// TIA Portal project "Donanım_Kesmesi_Uygulaması_V1" (V16)
// Vorlageprojekt für das Buch mit Zielsystem S7-1200

(* hardware
DEVICE "S7-1200-Station_1"  S7-1200 Station
   slot 0: "Baugruppenträger_0"  Rack  V1.0
   slot 1: "PLC_1"  CPU 1214C DC/DC/DC  6ES7 214-1AG40-0XB0  V4.4
   slot 2: "DQ 16x24VDC_1"  SM 1222 DQ16 x 24VDC  6ES7 222-1BH32-0XB0  V2.0
   slot 3: "AQ 2x14BIT_1"  SM 1232 AQ2  6ES7 232-4HB32-0XB0  V2.1
*)

// ===== PLC "PLC_1"  CPU 1214C DC/DC/DC =====

VAR_GLOBAL   // PLC tag table "Standard-Variablentabelle"
   "Sistem_Start_Mem." AT %M10.0 : Bool;
   "Kenar_Darbesi_1" AT %M20.0 : Bool;
   "Kenar_Darbesi_2" AT %M20.1 : Bool;
   "Kenar_Darbesi_3" AT %M20.2 : Bool;
   "Ürün_Sayısı" AT %MW30 : Int;
END_VAR

VAR_GLOBAL   // PLC tag table "Inputs"
   "Start_But" AT %I0.0 : Bool;
   "Stop_But" AT %I0.1 : Bool;
   "Acil_Stop_But" AT %I0.2 : Bool;
   "Sensör_!" AT %I0.3 : Bool;
   "Sensör_2" AT %I0.4 : Bool;
   "Sensör_3" AT %I0.5 : Bool;
END_VAR

VAR_GLOBAL   // PLC tag table "Outputs"
   "Durdurma_Kanalı" AT %Q0.0 : Bool;
   "Sayıcı_Ekranı" AT %QW30 : Int;
   "Konveyör_1" AT %QW32 : Int;
   "Konveyör_2" AT %QW34 : Int;
END_VAR

// folder: System blocks/Program resources

DATA_BLOCK "Tımer_1"   // DB1
{ S7_Optimized_Access := 'TRUE' }
AUTHOR : Simatic
FAMILY : IEC
NAME : IEC_TMR
VERSION : 1.0
// stored: InstanceOfName IEC_TIMER
"IEC_TIMER"
BEGIN
END_DATA_BLOCK

// folder: (top level)

FUNCTION "MHJ-PLC-Lab-Function-S71200" : Void   // FC9000, SCL
{ S7_Optimized_Access := 'TRUE' }
VERSION : 0.1
   VAR_TEMP
      rdTimeReturn : Int;
      outputTime : DTL;
      SyncVal : Byte;
      forVal : Int;
      forVal_2 : Int;
      Value : Byte;
   END_VAR
   VAR CONSTANT
      CompVal : Byte := 16#34;
      Value_01 : Byte := 16#11;
      Value_01_DW : DWord := 16#A165_D992;
      Value_02_DW : DWord := 16#58BE_4401;
   END_VAR
BEGIN

   #Value:=PEEK(area := 16#82,
        dbNumber := 0,
        byteOffset := 511);
   #Value := #Value + 1;

   POKE(area := 16#82,
        dbNumber := 0,
        byteOffset := 511,
        value := #Value);

   POKE(area:=16#81,
        dbNumber:=0,
        byteOffset:=1016,
        value:=#Value_01_DW);
   POKE(area := 16#81,
        dbNumber := 0,
        byteOffset := 1020,
        value := #Value_02_DW);

   POKE(area := 16#81,
        dbNumber := 0,
        byteOffset := 511,
        value := B#16#00);

   FOR #forVal := 0 TO 120 DO
       FOR #forVal_2:=0 TO 10 DO
           #rdTimeReturn:=RD_SYS_T(#outputTime);
           #rdTimeReturn := WR_SYS_T(#outputTime);
           #rdTimeReturn := RD_SYS_T(#outputTime);
           #rdTimeReturn := WR_SYS_T(#outputTime);
       END_FOR;
       #SyncVal:= PEEK(area := 16#81,
                      dbNumber := 0,
                      byteOffset := 511);
       IF #SyncVal = #CompVal THEN
          GOTO M_1;
       END_IF;
   END_FOR;
   RETURN;

   M_1:
   POKE(area := 16#81,
        dbNumber := 0,
        byteOffset := 511,
        value := B#16#0);
END_FUNCTION

ORGANIZATION_BLOCK "Main"   // OB1, LAD, ProgramCycle
TITLE = "Main Program Sweep (Cycle)"
{ S7_Optimized_Access := 'TRUE' }
VERSION : 0.1
   VAR_INPUT
      Initial_Call : Bool;   // Initial call of this OB
      Remanence : Bool;   // =True, if remanent data are available
   END_VAR
   VAR_TEMP   // added for the SCL form of the ladder/FBD networks
      _w1 : Bool;
      _w2 : Bool;
   END_VAR
BEGIN

REGION Network 1: Konnektierungsbaustein für PLC-Lab
   // Im Netzwerk 1 wird der Konnektierungsbaustein für PLC-Lab aufgerufen.
   // Dieser Aufruf darf nicht entfernt werden!
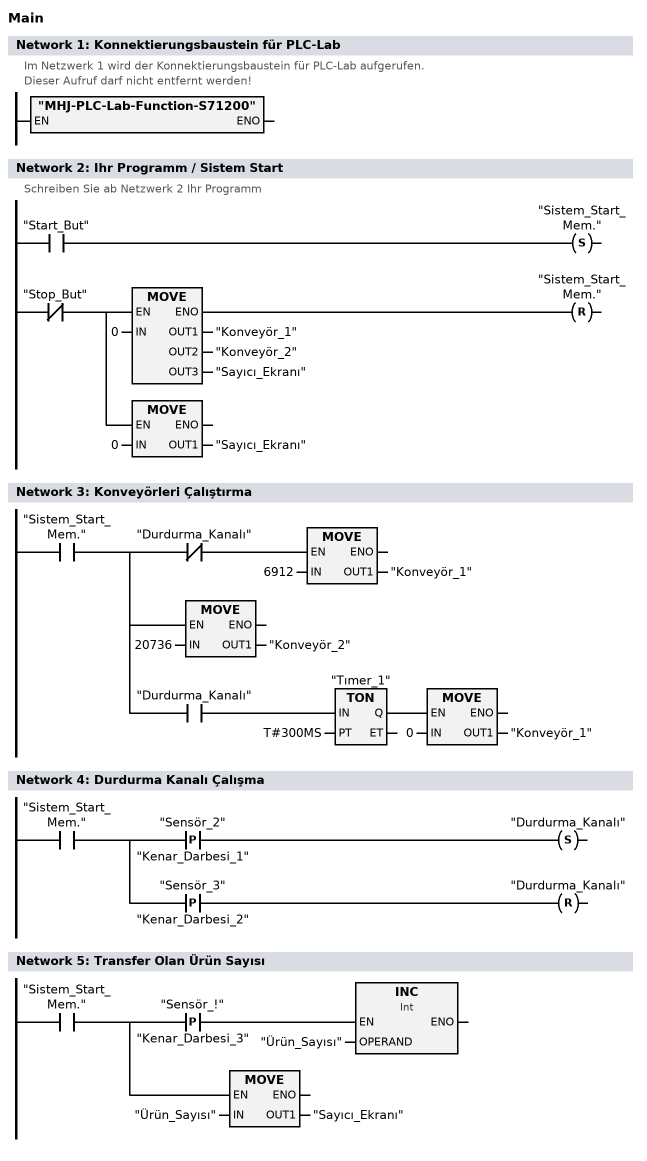
   RUNG wire#powerrail
      "MHJ-PLC-Lab-Function-S71200"()
   END_RUNG
   // the same network as SCL:
   "MHJ-PLC-Lab-Function-S71200"();
END_REGION

REGION Network 2: Ihr Programm / Sistem Start
   // Schreiben Sie ab Netzwerk 2 Ihr Programm
   RUNG wire#powerrail
      Contact( "Start_But" )
      S_Coil( "Sistem_Start_Mem." )
   END_RUNG
   RUNG wire#powerrail
      I_Contact( "Stop_But" )
      wire#w1
      Move(in := 0, out1 => "Konveyör_1", out2 => "Konveyör_2", out3 => "Sayıcı_Ekranı")
      R_Coil( "Sistem_Start_Mem." )
   END_RUNG
   RUNG wire#w1
      Move(in := 0, out1 => "Sayıcı_Ekranı")
   END_RUNG
   // the same network as SCL:
   IF "Start_But" THEN "Sistem_Start_Mem." := TRUE; END_IF;
   IF NOT "Stop_But" THEN
       "Konveyör_1" := 0;
       "Konveyör_2" := 0;
       "Sayıcı_Ekranı" := 0;
       "Sistem_Start_Mem." := FALSE;
       "Sayıcı_Ekranı" := 0;
   END_IF;
END_REGION

REGION Network 3: Konveyörleri Çalıştırma
   IF "Sistem_Start_Mem." AND NOT "Durdurma_Kanalı" THEN "Konveyör_1" := 6912; END_IF;
   IF "Sistem_Start_Mem." THEN "Konveyör_2" := 20736; END_IF;
   "Tımer_1".TON(IN := "Sistem_Start_Mem." AND "Durdurma_Kanalı", PT := T#300MS);
   IF "Tımer_1".Q THEN "Konveyör_1" := 0; END_IF;
END_REGION

REGION Network 4: Durdurma Kanalı Çalışma
   RUNG wire#powerrail
      Contact( "Sistem_Start_Mem." )
      wire#w1
      P_Contact(operand := "Sensör_2", bit := "Kenar_Darbesi_1")
      S_Coil( "Durdurma_Kanalı" )
   END_RUNG
   RUNG wire#w1
      P_Contact(operand := "Sensör_3", bit := "Kenar_Darbesi_2")
      R_Coil( "Durdurma_Kanalı" )
   END_RUNG
   // the same network as SCL:
   #_w1 := "Sistem_Start_Mem." AND "Sensör_2" AND NOT "Kenar_Darbesi_1";   // rising edge of "Sensör_2"
   "Kenar_Darbesi_1" := "Sensör_2";
   IF #_w1 THEN "Durdurma_Kanalı" := TRUE; END_IF;
   #_w2 := "Sistem_Start_Mem." AND "Sensör_3" AND NOT "Kenar_Darbesi_2";   // rising edge of "Sensör_3"
   "Kenar_Darbesi_2" := "Sensör_3";
   IF #_w2 THEN "Durdurma_Kanalı" := FALSE; END_IF;
END_REGION

REGION Network 5: Transfer Olan Ürün Sayısı
   RUNG wire#powerrail
      Contact( "Sistem_Start_Mem." )
      wire#w1
      P_Contact(operand := "Sensör_!", bit := "Kenar_Darbesi_3")
      { S7_Templates := "DestType := Int" } Inc( "Ürün_Sayısı" )
   END_RUNG
   RUNG wire#w1
      Move(in := "Ürün_Sayısı", out1 => "Sayıcı_Ekranı")
   END_RUNG
   // the same network as SCL:
   #_w1 := "Sistem_Start_Mem." AND "Sensör_!" AND NOT "Kenar_Darbesi_3";   // rising edge of "Sensör_!"
   "Kenar_Darbesi_3" := "Sensör_!";
   IF #_w1 THEN "Ürün_Sayısı" := "Ürün_Sayısı" + 1; END_IF;
   IF "Sistem_Start_Mem." THEN "Sayıcı_Ekranı" := "Ürün_Sayısı"; END_IF;
END_REGION
END_ORGANIZATION_BLOCK

ORGANIZATION_BLOCK "Acil Stop Kesme"   // OB40, LAD, HWProcessInterrupt
{ S7_Optimized_Access := 'TRUE' }
VERSION : 0.1
   VAR_INPUT
      LADDR : Hw_Io;   // Hardware identifier
      USI : Word;   // User structure identifier
      IChannel : USInt;   // Interrupt channel number
      EventType : Byte;   // EventType
   END_VAR
   VAR_TEMP   // added for the SCL form of the ladder/FBD networks
      _w1 : Bool;
   END_VAR
BEGIN

REGION Network 1: Acil Stop Programı
   // - Donanım kesmesi, bir sensör girişinde yükselen veya düşen kenar oluştuğu anda OB1’i beklemeden ilgili kesme OB’sini çalıştırır ve sahada hızlı sensör/HSC olaylarında bu şekilde kullanılır; ancak eğitimdeki acil stop örneği sadece öğretim amaçlıdır, gerçek acil stop emniyet rölesi veya F-CPU ile yapılmalıdır.
   // -  OB40 makineye “dur” komutu verir; emniyet rölesi veya F sistemi ise makinenin gerçekten güvenli şekilde durmasını garanti eden asıl yapıdır.
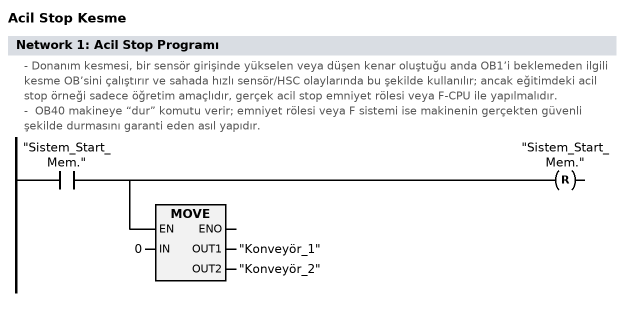
   RUNG wire#powerrail
      Contact( "Sistem_Start_Mem." )
      wire#w1
      R_Coil( "Sistem_Start_Mem." )
   END_RUNG
   RUNG wire#w1
      Move(in := 0, out1 => "Konveyör_1", out2 => "Konveyör_2")
   END_RUNG
   // the same network as SCL:
   #_w1 := "Sistem_Start_Mem.";
   IF #_w1 THEN
       "Sistem_Start_Mem." := FALSE;
       "Konveyör_1" := 0;
       "Konveyör_2" := 0;
   END_IF;
END_REGION
END_ORGANIZATION_BLOCK